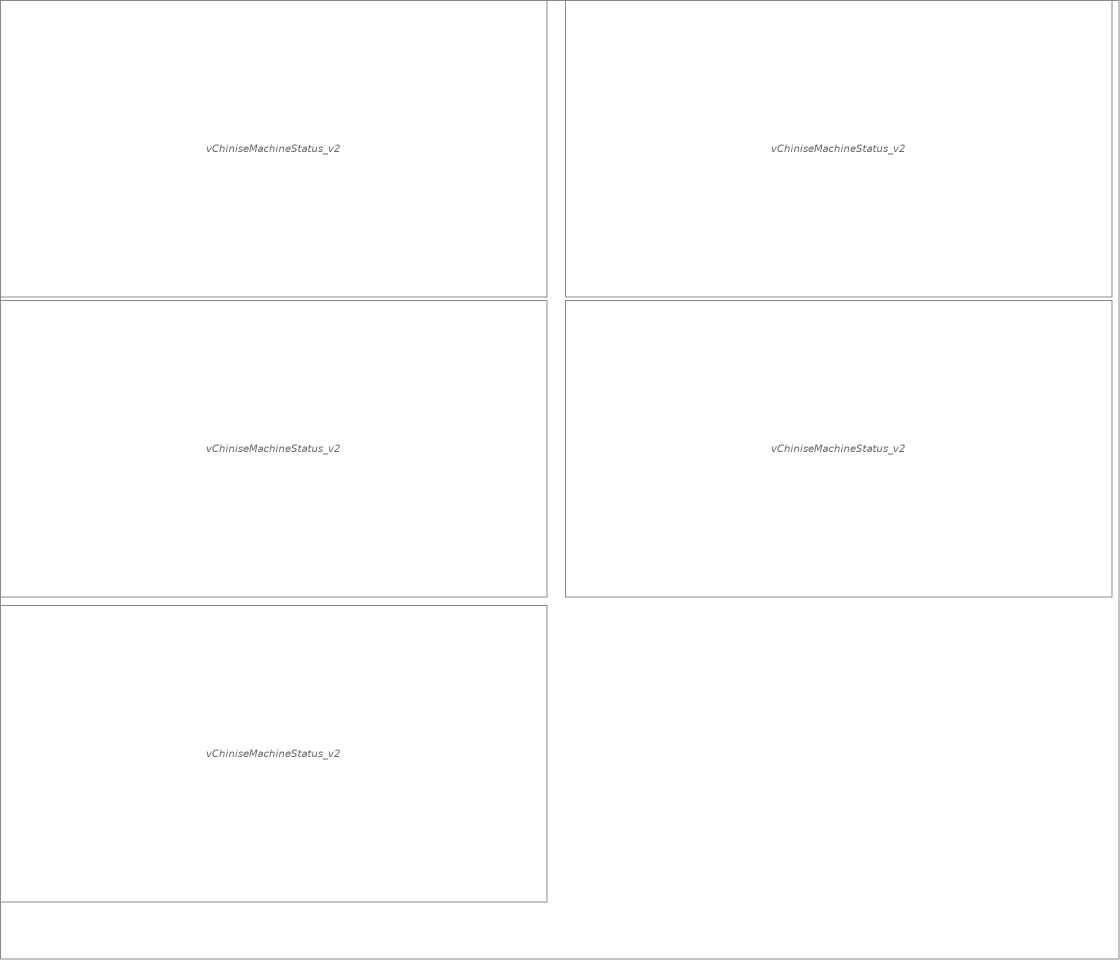
VISUALIZATION vFillingLine  // 1120x960
    Frame (0,0 547x297)
        shows vChiniseMachineStatus_v2(stData := MAIN.fb_Filler_A_Machine.stHMI, stParams := GVL.st_Filler_A_Parameters)
    Frame (0,300 547x297)
        shows vChiniseMachineStatus_v2(stData := MAIN.fb_Cork_Machine.stHMI, stParams := GVL.st_Cork_Parameters)
    Frame (565,0 547x297)
        shows vChiniseMachineStatus_v2(stData := MAIN.fb_Sticker_Machine.stHMI, stParams := GVL.st_Sticker_Parameters)
    Frame (565,300 547x297)
        shows vChiniseMachineStatus_v2(stData := MAIN.fb_Laser_Machine.stHMI, stParams := GVL.st_Laser_Parameters)
    Frame (0,605 547x297)
        shows vChiniseMachineStatus_v2(stData := MAIN.fb_Filler_B_Machine.stHMI, stParams := GVL.st_Filler_B_Parameters)
END_VISUALIZATION

(* stored: Version 1.1.0.1, ProductVersion 3.1.4024.13
   Visu vFillingLine: Id {2def58da-3738-4b48-9b70-f9aa63ccdbb3} *)
